(* CODESYS project ApplicationManager.project
   Description: The use of the system library, “CmpApp” is demonstrated. Information about the project and application are retrieved as well as area addresses and sizes of the different data types. It is also possible to stop or reset an application within a program.
   Title: Application Manager

Project tree, tasks and I/O mapping:
  Device : CODESYS Control Win V3 x64, 3S - Smart Software Solutions GmbH, version 3.5.15.0
    application App1
      libraries: CmpApp, 3.4.3.0 (System); CAA File, 3.4.3.0 (CAA Technical Workgroup); SysTypes Interfaces, * (System)
      task MainTask (cyclic, interval t#20ms, priority 1) calls Main
      program AppInteract [ST]
      function block ExceptionDuring_InitCode [ST]: FB_Init
      program AppInfo [ST]
      program AppRetain [ST]
      program Main [ST]
      program AppAreas [ST]
      global variables RetainPersistent
      license
    application App2
      libraries: CmpApp, 3.4.3.0 (System); SysTypes Interfaces, * (System)
      task MainTask (cyclic, interval t#20ms, priority 1) calls PLC_PRG
      program PLC_PRG [ST]
      license
  00000000-0000-0000-0000-000000000000|C:\Users\m.lamp\Documents\license.txt
*)

// Device/App1/RetainPersistent
VAR_GLOBAL PERSISTENT RETAIN
	byByte      : BYTE   := 255;
	wWord       : WORD   := 65535;
	dwDWord     : DWORD  := 4294967295;
	siINT       : SINT   := 127;
	usiINT      : USINT  := 255;
	iINT        : INT    := 32767;
	uiUInt      : UINT   := 65535;
	diDInt      : DINT   := 2147483647;
	udiUDInt    : UDINT  := 4294967295;
	rReal       : REAL   := 5.5;
	rLREAL      : LREAL  := 7.897;
	bGreen      : BOOL   := FALSE;
	dDate       : DATE   := D#1980-01-01;
	tTime       : TIME   := T#2ms;
	dtDt        : DT     := DT#1980-01-01-01:01:01;
	todTOD      : TOD    := TOD#01:01:01.001;
END_VAR

// Device/App1/Main
PROGRAM Main
VAR
	(*Uncomment it to generate an exception. *) 
	//fbException : ExceptionDuring_InitCode;
END_VAR

(* Application information *)
AppInfo();

(* Information about areas *)
AppAreas();

(* restore and restore retain variables *)
AppRetain();

(* Application interactions, like start, stop, reset etc. *)
AppInteract();

END_PROGRAM

// Device/App1/AppInfo
PROGRAM AppInfo
VAR
	apApps			: ARRAY[0..1] OF POINTER TO APPLICATION; (* Array for both application *)
	sAppName 		: STRING := 'App2';
	pAppByName		: POINTER TO APPLICATION;
	pApp			: POINTER TO APPLICATION;
	pCurrentApp		: POINTER TO APPLICATION;
	pAppInfo		: POINTER TO APPLICATION_INFO;
	pProjectInfo	: POINTER TO PROJECT_INFO; (* Pointer to project information *)
	Result			: RTS_IEC_RESULT; (* Error codes of the different funciton *)
	udiNumSessions	: UDINT; (* Number of active sessions *)
	iAppCnt			: INT; (* Number of applicatinos. *)
END_VAR

(* This program retrieves several information about the current application and the project
   as well as the number of active sessions. *)

(* Iterate through all Applications and save them in an array. *)
pApp := AppGetFirstApp(pResult := ADR(Result));

WHILE pApp <> 0 DO
	apApps[iAppCnt] := pApp;
	pApp := AppGetNextApp(pApp, pResult := ADR(Result));
END_WHILE

(* Get the current Application. *)
pCurrentApp := AppGetCurrent(pResult := ADR(Result));

(* Get an Application with the corresponding name *)
pAppByName := AppFindApplicationByName(sAppName, ADR(Result));

(* Fetch some application information *)
pAppInfo := AppGetApplicationInfo(pCurrentApp, ADR(Result));

(* Fetch the project information *)
Result := AppGetProjectInformation(pCurrentApp, pProjectInfo);

(* get the active sessions of the application *)
Result := AppNumOfActiveSessions(pCurrentApp, ADR(udiNumSessions));

END_PROGRAM

// Device/App1/AppAreas
PROGRAM AppAreas
VAR
	iCounter 				: INT;
	pApp					: POINTER TO APPLICATION;
	Result					: RTS_IEC_RESULT;
	pbyCodeAreaAddress 		: POINTER TO BYTE;
	pbyDataAreaAddress 		: POINTER TO BYTE;
	pbyRetainAreaAddress 	: POINTER TO BYTE;
	pbyInputAreaAddress 	: POINTER TO BYTE;
	pbyOutputAreaAddress 	: POINTER TO BYTE;
	
	udiCodeAreaSize			: __XWORD;
	udiDataAreaSize			: __XWORD;
	udiRetainAreaSize		: __XWORD;
	udiInputAreaSize		: __XWORD;
	udiOutputAreaSize		: __XWORD;
	
	pbyCodeSegmentAddress	: POINTER TO BYTE;
	pbyCodeSegmentSize		: __XWORD;
END_VAR

VAR CONSTANT
	cTest : INT := 4;
END_VAR

(* This program retrieves area addresses and sizes of five different data types. *)
iCounter := iCounter + 1;

(* Get the Application with the help of a variable. *)
pApp := AppGetApplicationByAreaAddress(ADR(iCounter));

(* For the area types see CmpApp library --> AreaTypes *)
pbyCodeAreaAddress := AppGetAreaAddress(pApp, AreaTypes.DA_CODE, ADR(Result));
pbyDataAreaAddress := AppGetAreaAddress(pApp, AreaTypes.DA_DATA, ADR(Result));
pbyRetainAreaAddress := AppGetAreaAddress(pApp, AreaTypes.DA_RETAIN, ADR(Result));
pbyInputAreaAddress := AppGetAreaAddress(pApp, AreaTypes.DA_INPUT, ADR(Result));
pbyOutputAreaAddress := AppGetAreaAddress(pApp, AreaTypes.DA_OUTPUT, ADR(Result));

(* Retrieve the size of the areas. *)
udiCodeAreaSize := AppGetAreaSize(pApp, AreaTypes.DA_CODE, ADR(Result));
udiDataAreaSize := AppGetAreaSize(pApp, AreaTypes.DA_DATA, ADR(Result));
udiRetainAreaSize := AppGetAreaSize(pApp, AreaTypes.DA_RETAIN, ADR(Result));
udiInputAreaSize := AppGetAreaSize(pApp, AreaTypes.DA_INPUT, ADR(Result));
udiOutputAreaSize := AppGetAreaSize(pApp, AreaTypes.DA_OUTPUT, ADR(Result));


(* Get the segment address and size, which are within a area. *)
pbyCodeSegmentAddress := AppGetSegmentAddress(pApp, AreaTypes.DA_INPUT, ADR(Result));
pbyCodeSegmentSize := AppGetSegmentSize(pApp, AreaTypes.DA_INPUT, ADR(Result));

END_PROGRAM

// Device/App1/AppRetain
PROGRAM AppRetain

VAR
	fbDelete            : FILE.Delete; (* Function block to delete the file *)
    (* The retain file <application-name>.ret is placed in the directory of the bootproject *)
	sFileName           : STRING := 'App1.ret';
	pApp				: POINTER TO APPLICATION;
	Result              : RTS_IEC_RESULT; (* Result code *)
	xInit				: BOOL;
END_VAR

(* The retain variables are stores in a file and get retrieved afterwards. *)
IF NOT xInit THEN
	
	(* First delete the retain file.
	   This is necessary, because the function AppStoreRetainsInFile appends the data at the end of the file. *)
	fbDelete(xExecute:=TRUE, sFileName:=sFileName);
	IF fbDelete.xDone OR (fbDelete.xError AND fbDelete.eError = FILE.ERROR.NOT_EXIST) THEN
		(* Attention: It takes at least one cycle until xDone is TRUE *)
		fbDelete(xExecute:=FALSE);
		xInit := TRUE;
		(* Now, it's the time to save the retains. *)
		pApp := AppGetCurrent(pResult:=ADR(Result));
		IF pApp <> 0 THEN
			(* Store the variables in a file*)
			Result := AppStoreRetainsInFile(pApp,sFileName);
		END_IF
	END_IF
END_IF

(* Restore the Retain Variables from the file.
   For storing and restoring, the same pointer to application (pApp) must be used.*)
Result := AppRestoreRetainsFromFile(pApp, sFileName);

END_PROGRAM

// Device/App1/AppInteract
PROGRAM AppInteract
VAR
	pApp		: POINTER TO APPLICATION;
	Result		: RTS_IEC_RESULT;
	sApp2		: STRING := 'App2';
	xStart		: BOOL; (* Start the application. *)
	xStop		: BOOL; (* Stop the application. *)
	xResetWarm	: BOOL; (* Do a reset warm *)
	xResetCold	: BOOL; (* Do a reset cold. *)
	xResetOrigin: BOOL; (* Do a reset origin. *)
END_VAR

(* This programs shows interaction possibilities on a task. All interactions are done at
   the App2 application. *)

pApp := AppFindApplicationByName(sApp2, ADR(Result));

(* start App2 *)
IF xStart THEN
	xStart := FALSE;
	Result := AppStartApplication(pApp);
END_IF

(* stop App2 *)
IF xStop THEN
	xStop := FALSE;
	Result := AppStopApplication(pApp);
END_IF

(* reset warm on App2 *)
IF xResetWarm THEN
	xResetWarm := FALSE;
	Result := AppReset(pApp, RESET_OPTION.RTS_RESET);
END_IF

(* reset cold on App2 *)
IF xResetCold THEN
	xResetCold := FALSE;
	Result := AppReset(pApp, RESET_OPTION.RTS_RESET_COLD);
END_IF

(* reset origin on App2 *)
IF xResetOrigin THEN
	xResetOrigin := FALSE;
	Result := AppReset(pApp, RESET_OPTION.RTS_RESET_ORIGIN);
END_IF

END_PROGRAM

// Device/App1/ExceptionDuring_InitCode
FUNCTION_BLOCK ExceptionDuring_InitCode
VAR_INPUT
END_VAR
VAR_OUTPUT
END_VAR
VAR
	Result : RTS_IEC_RESULT;
END_VAR

METHOD FB_Init : BOOL
VAR_INPUT
	bInitRetains: BOOL;
	bInCopyCode: BOOL;	
END_VAR
VAR
	pApp : POINTER TO APPLICATION;
END_VAR
pApp := AppGetCurrent(ADR(Result));

(* Exception code "Application is running on wrong target". Can be used for library protection! *)
Result := AppGenerateException(pApp:=pApp, ulException:=Exception.RTSEXCPT_APP_TARGET_MISMATCH);
END_METHOD

END_FUNCTION_BLOCK

// Device/App2/PLC_PRG
PROGRAM PLC_PRG
VAR
	uiApp2Counter	: UINT;
END_VAR

(* Counter to see when this application is stopped from 'App1' *)
uiApp2Counter := uiApp2Counter + 1;

END_PROGRAM
